TYPE ref_ele_param :
STRUCT
	var_mutex : INT;
	var_timeOut : TIME;
	flg_reset :BOOL;
END_STRUCT
END_TYPE

(* stored: Version 1.1.0.1, ProductVersion 3.1.4024.11
   DUT ref_ele_param: Id {61031c65-d6c0-4664-91e5-59d2c61ed546} *)
